// TIA Portal V17 export
// export: Created 2022-07-20T06:59:45.0934142Z, ExportSetting WithDefaults, DisplayName Totally Integrated Automation Portal, DisplayVersion V17, DisplayName TIA Portal Openness, DisplayVersion V17, DisplayName TIA Portal Version Control Interface, DisplayVersion V17, DisplayName SINAMICS Startdrive Advanced, DisplayVersion V17, DisplayName SINAMICS Startdrive G130, G150, S120, S150, SINAMICS MV, S210, DisplayVersion V17, DisplayName SINAMICS Startdrive G110M, G120, G120C, G120D, G120P, G115D, DisplayVersion V17, DisplayName STEP 7 Professional, DisplayVersion V17, DisplayName STEP 7 Safety, DisplayVersion V17, DisplayName WinCC Advanced, DisplayVersion V17
FUNCTION_BLOCK "FB10090_LampIRControl"   // FB10090, LAD
TITLE = FB10090_LampIRControl
{ S7_Optimized_Access := 'TRUE' }
AUTHOR : Jonathan
FAMILY : 1009x_DRYER_IR
VERSION : 1.0
// Release note : 
// 1.0 - Feature developped
// stored: AutoNumber false, IsIECCheckEnabled false, IsRetainMemResEnabled false, MemoryReserve 100, SetENOAutomatically false, UDAEnableTagReadback false
   VAR_INPUT
      EnableModule : Bool;
      PowerOK : Bool;
      StartLampCommand : Bool;
      PowerSetpoint : Real;   // (0-100%)
      ThermalContatorOk : Bool;
      PowerSupplyAlarm : Bool;
   END_VAR
   VAR_OUTPUT
      AnalogPowerValue : Int;
      ActivePowerRelay : Bool;
   END_VAR
BEGIN

REGION Network 1: Active power relay
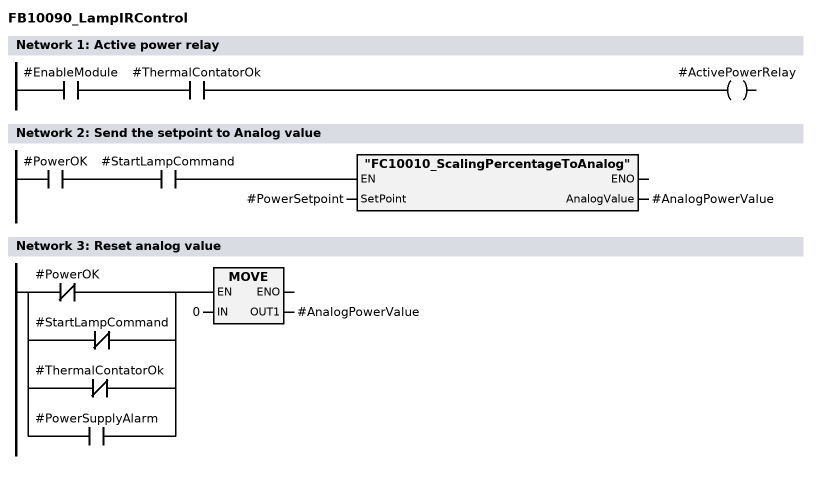
   RUNG wire#powerrail
      Contact( #EnableModule )
      Contact( #ThermalContatorOk )
      Coil( #ActivePowerRelay )
   END_RUNG
   // the same network as SCL:
   #ActivePowerRelay := #EnableModule AND #ThermalContatorOk;
END_REGION

REGION Network 2: Send the setpoint to Analog value
   RUNG wire#powerrail
      Contact( #PowerOK )
      Contact( #StartLampCommand )
      "FC10010_ScalingPercentageToAnalog"(SetPoint := #PowerSetpoint, AnalogValue => #AnalogPowerValue)
   END_RUNG
   // the same network as SCL:
   IF #PowerOK AND #StartLampCommand THEN
       "FC10010_ScalingPercentageToAnalog"(SetPoint := #PowerSetpoint, AnalogValue => #AnalogPowerValue);
   END_IF;
END_REGION

REGION Network 3: Reset analog value
   RUNG wire#powerrail
      I_Contact( #PowerOK )
      wire#w1
      { S7_GenerateENO := "TRUE" } Move(in := 0, out1 => #AnalogPowerValue)
   END_RUNG
   RUNG wire#powerrail
      I_Contact( #StartLampCommand )
   END_RUNG wire#w1
   RUNG wire#powerrail
      I_Contact( #ThermalContatorOk )
   END_RUNG wire#w1
   RUNG wire#powerrail
      Contact( #PowerSupplyAlarm )
   END_RUNG wire#w1
   // the same network as SCL:
   IF NOT #PowerOK OR NOT #StartLampCommand OR NOT #ThermalContatorOk OR #PowerSupplyAlarm THEN
       #AnalogPowerValue := 0;
   END_IF;
END_REGION
END_FUNCTION_BLOCK
